FUNCTION_BLOCK ButtonDs
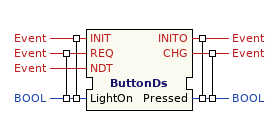
  EVENT_INPUT
    INIT WITH LightOn;
    REQ WITH LightOn;
    NDT;
  END_EVENT
  EVENT_OUTPUT
    INITO WITH Pressed;
    CHG WITH Pressed;
  END_EVENT
  VAR_INPUT
    LightOn : BOOL;
  END_VAR
  VAR_OUTPUT
    Pressed : BOOL;
  END_VAR
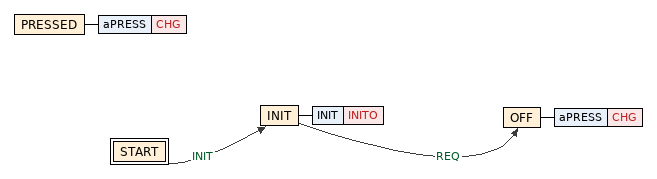
  EC_STATES
    START;
    INIT : INIT -> INITO;
    OFF : aPRESS -> CHG;
    PRESSED : aPRESS -> CHG;
  END_STATES
  EC_TRANSITIONS
    START TO INIT := INIT;
    INIT TO OFF := REQ;
  END_TRANSITIONS
  ALGORITHM INIT IN ST:
Pressed := FALSE;
  END_ALGORITHM
  ALGORITHM aOFF IN ST:
Pressed := FALSE;
  END_ALGORITHM
  ALGORITHM aPRESS IN ST:
Pressed := TRUE;
  END_ALGORITHM
END_FUNCTION_BLOCK
